PROGRAM Pneumatics_Template
VAR
END_VAR

//Test the program to control pneumatic acutator through PneumaticsVisu.
//Currently implemented control of single solenoid through PLC and and manually, with two momentary push buttons.

(*
The number of axis is already set to one, don't chnage the Pneumatic Axis Selection.
Default mode of control is SINGLE_SOLENOID_PLC.
Activate the Permit signal through bPermit button.

Simulate the position of actuator through bLimitBwd and bLimitFwd buttons.
When bLimitBwd := TRUE, cylinder is retracted, when bLimitFwd := TRUE, cylinder is extracted, when bLimitBwd := FALSE
and bLimitFwd := FALSE, cylinder is moving.

Write allowed times for extending and retracting the cylinder in seconds in nTimeToExtend and nTimeToRetract.

Use the buttons StartExtend and StartRetract to control the cylider, based on the selected mode SINGLE_SOLENOID_PLC and SINGLE_SOLENOID_MANUAL.

To simulate errors:
- Leave bLimitFwd activated until the allowed time elapses when moving forward.
- Leave bLimitBwd activated until allowed time elapses when moving backward.
- Deactivate both limit switches and leave the allowed time to elapse.
- Deactivate bPermit while the cylnder is moving. Cylinder can't move if the bPermit := FALSE.
- Reset errors with bReset button, and choose the wanted mode again.
*)

END_PROGRAM

(* stored: Version 1.1.0.1, ProductVersion 3.1.4024.5
   POU Pneumatics_Template: Id {7bf401fb-a600-4741-a67b-36f20e194cfc}, SpecialFunc None *)
